VAR_GLOBAL

	eMachineState					: E_MachineState;
	UI_EnableHighSpeed				: BOOL;
END_VAR

(* stored: Version 1.1.0.1, ProductVersion 3.1.4024.9
   GVL GVL: Id {bbef5aca-9751-4345-a16a-b08174c7e4ef} *)
